// TIA Portal V18 export
FUNCTION_BLOCK "LIVE_BLINK_MONITOR_TESTER"   // FB66, FBD
{ S7_Optimized_Access := 'TRUE' }
VERSION : 0.1
// stored: AutoNumber true, IsIECCheckEnabled false, IsRetainMemResEnabled false, MemoryReserve 100, SetENOAutomatically false, UDAEnableTagReadback false
   VAR_OUTPUT
      flashing : Bool;
      high : Bool;
   END_VAR
   VAR
      BLINKER_Instance { S7_SetPoint := 'True'} : "BLINKER";
      run : Bool;
      blink_t_on : Time;
      blink_t_off : Time;
      run_t_on : Time;
      run_t_off : Time;
      blink_run { S7_SetPoint := 'True'} : "BLINKER";
      test_problems : Bool;
   END_VAR
BEGIN

REGION Network 1
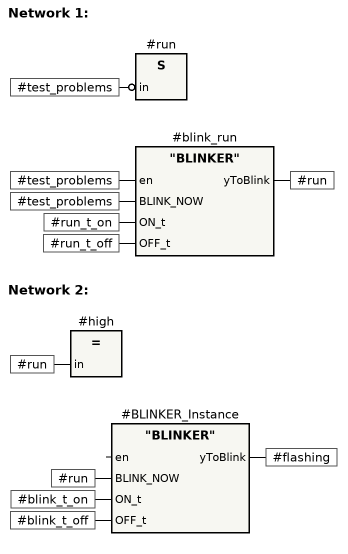
   IF NOT #test_problems THEN #run := TRUE; END_IF;
   IF #test_problems THEN
       #blink_run(BLINK_NOW := #test_problems, ON_t := #run_t_on, OFF_t := #run_t_off, yToBlink => #run);   // "BLINKER"
   END_IF;
END_REGION

REGION Network 2
   #high := #run;
   #BLINKER_Instance(BLINK_NOW := #run, ON_t := #blink_t_on, OFF_t := #blink_t_off, yToBlink => #flashing);   // "BLINKER"
END_REGION
END_FUNCTION_BLOCK
